Staubli VAL3: debug.pgx

public program debug(num& x_nExecStatus)
begin

  // Do nothing
  // See start() program for more details

end
